(* LS Electric XG5000 project: CMore_ModTCP *)
(* PLC LSPLC *)
(* module base 0 slot 0: Input/Output Module:XEM-DN/DP32HP (DC 24V Input, Transistor Output, 32 Contacts) *)
(* module base 0 slot 1: Internal Positioning:XBF-PO06E (Open Collector Type, 6 Axis) *)

PROGRAM NewProgram (* task: Scan Program *)
VAR
    BOOL_FROM_HMI AT %MX6416 : BOOL;
    BOOL_TO_HMI AT %MX3216 : BOOL;
    DINT_FROM_HMI AT %MD804 : DINT;
    DINT_TO_HMI AT %MD304 : DINT;
    DWORD_FROM_HMI AT %MD307 : DWORD;
    DWORD_TO_HMI AT %MD807 : DWORD;
    INT_FROM_HMI AT %MW1600 : INT;
    INT_TO_HMI AT %MW600 : INT;
    REAL_FROM_HMI AT %MD806 : REAL;
    REAL_TO_HMI AT %MD306 : REAL;
    STRING_FROM_HMI AT %MW1616 : STRING;
    STRING_TO_HMI AT %MD308 : STRING;
    tempDINT : DINT;
    tempINT : INT;
    tempReal : REAL;
    tempUDINT : UDINT;
    tempUINT : UINT;
    Temp_Toggle : BOOL;
    UDINT_FROM_HMI AT %MD805 : UDINT;
    UDINT_TO_HMI AT %MD305 : UDINT;
    UINT_FROM_HMI AT %MW1601 : UINT;
    UINT_TO_HMI AT %MW601 : UINT;
    WORD_FROM_HMI AT %MW602 : WORD;
    WORD_TO_HMI AT %MW1602 : WORD;
END_VAR

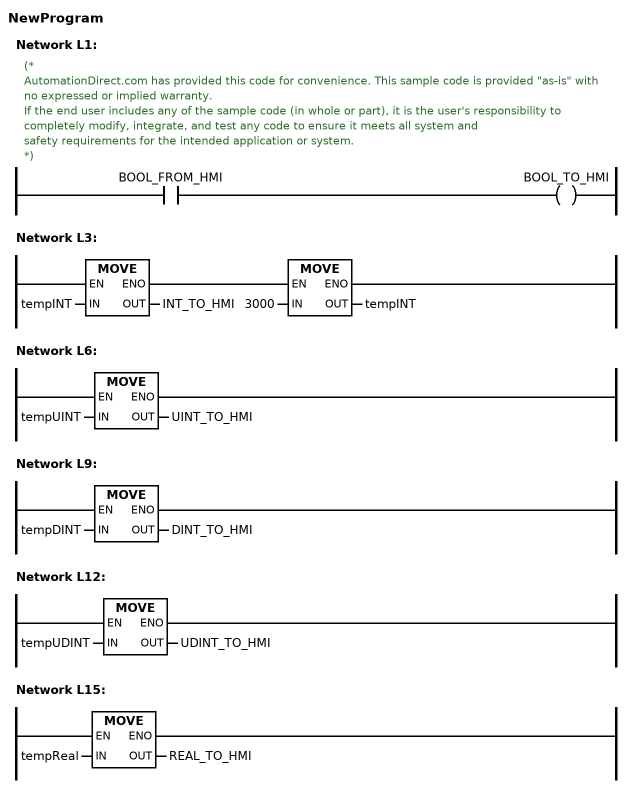
(* ( * / AutomationDirect.com has provided this code for convenience. This sample code is provided "as-is" with no expressed or implied warranty. / If the end user includes any of the sample code (in whole or part), it is the user's responsibility to completely modify, integrate, and test any code to ensure it meets all system and / safety requirements for the intended application or system. / * ) *)
(* Rung L1 *)
BOOL_TO_HMI := BOOL_FROM_HMI;
(* Rung L3 *)
INT_TO_HMI := tempINT;
tempINT := 3000;
(* Rung L6 *)
UINT_TO_HMI := tempUINT;
(* Rung L9 *)
DINT_TO_HMI := tempDINT;
(* Rung L12 *)
UDINT_TO_HMI := tempUDINT;
(* Rung L15 *)
REAL_TO_HMI := tempReal;
END_PROGRAM